Fanuc KAREL source: kt00761.KL

-- PROVISIONAL review KL for V940-1; original PC SHA256 b8ad44cf5acb5c369031780f7e9b712dce91da5a9206288c3336bd11b42e6d79
-- Incomplete behavior may be omitted. Consult companion uncertainty JSON. Do not deploy.
PROGRAM KT00761
%NOLOCKGROUP
VAR
  I1 : INTEGER
  I2 : INTEGER
  OUT : REAL
BEGIN
  -- V9_ZERO_TABLE_METADATA_HINT layout=0001; no indexed target words; source/name/runtime held
  -- UNRESOLVED_PC offsets 5-16; opcodes 2E,23
  -- UNRESOLVED_PC offsets 21-32; opcodes 2E,23
  -- UNRESOLVED_PC offsets 37-48; opcodes 2E,23
  -- UNRESOLVED_PC offsets 53-64; opcodes 2E,23
  -- UNRESOLVED_PC offsets 69-86; opcodes 27,27,21,64,76,23
  -- UNRESOLVED_PC offsets 91-95; opcodes 7F
END KT00761
